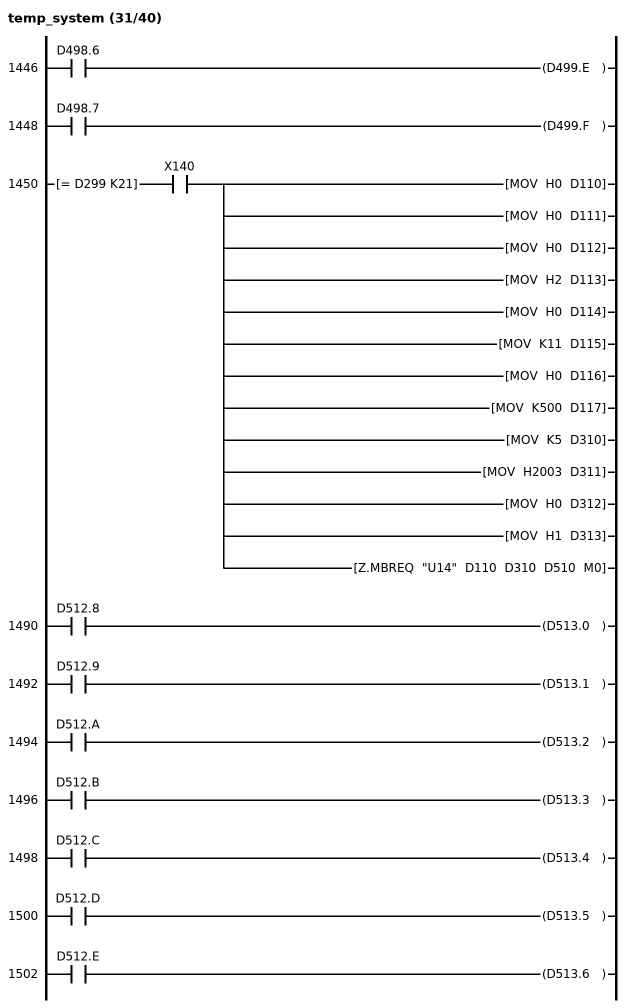
[picture p264: ladder of temp_system, rungs at steps 1446 to 1502]
1446  LD      D498.6
      OUT     D499.E
1448  LD      D498.7
      OUT     D499.F
1450  LD=     D299 K21
      AND     X140
      MOV     H0 D110
      MOV     H0 D111
      MOV     H0 D112
      MOV     H2 D113
      MOV     H0 D114
      MOV     K11 D115
      MOV     H0 D116
      MOV     K500 D117
      MOV     K5 D310
      MOV     H2003 D311
      MOV     H0 D312
      MOV     H1 D313
      Z.MBREQ "U14" D110 D310 D510 M0
1490  LD      D512.8
      OUT     D513.0
1492  LD      D512.9
      OUT     D513.1
1494  LD      D512.A
      OUT     D513.2
1496  LD      D512.B
      OUT     D513.3
1498  LD      D512.C
      OUT     D513.4
1500  LD      D512.D
      OUT     D513.5
1502  LD      D512.E
      OUT     D513.6
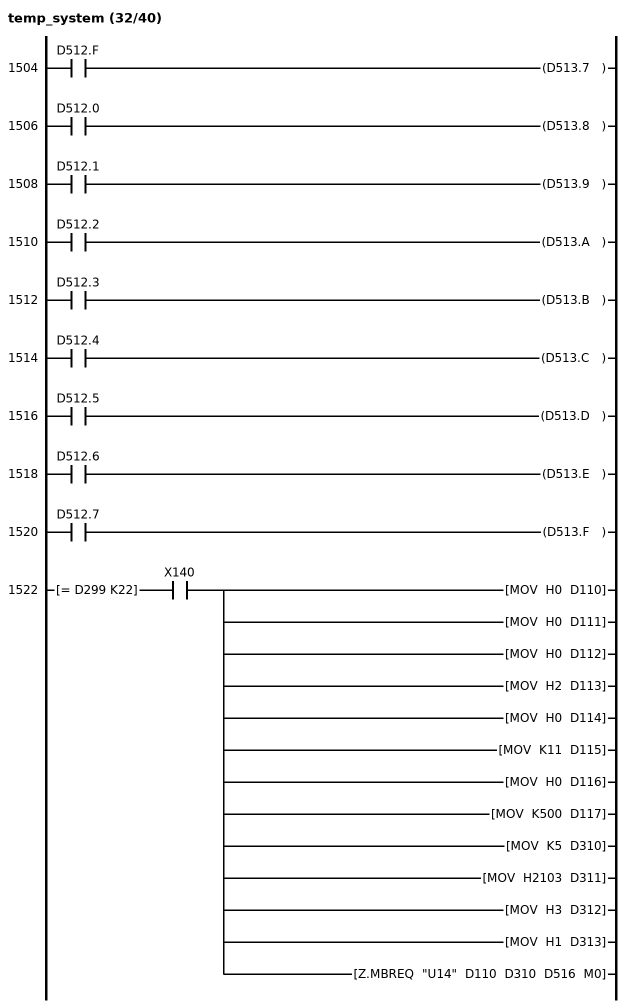
1504  LD      D512.F
      OUT     D513.7
1506  LD      D512.0
      OUT     D513.8
1508  LD      D512.1
      OUT     D513.9
1510  LD      D512.2
      OUT     D513.A
1512  LD      D512.3
      OUT     D513.B
1514  LD      D512.4
      OUT     D513.C
1516  LD      D512.5
      OUT     D513.D
1518  LD      D512.6
      OUT     D513.E
1520  LD      D512.7
      OUT     D513.F
1522  LD=     D299 K22
      AND     X140
      MOV     H0 D110
      MOV     H0 D111
      MOV     H0 D112
      MOV     H2 D113
      MOV     H0 D114
      MOV     K11 D115
      MOV     H0 D116
      MOV     K500 D117
      MOV     K5 D310
      MOV     H2103 D311
      MOV     H3 D312
      MOV     H1 D313
      Z.MBREQ "U14" D110 D310 D516 M0
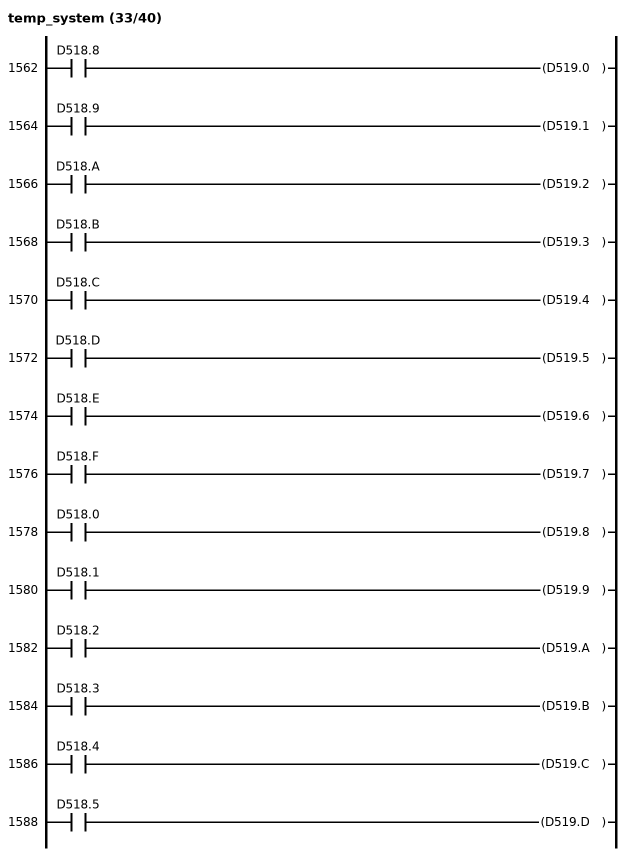
1562  LD      D518.8
      OUT     D519.0
1564  LD      D518.9
      OUT     D519.1
1566  LD      D518.A
      OUT     D519.2
1568  LD      D518.B
      OUT     D519.3
1570  LD      D518.C
      OUT     D519.4
1572  LD      D518.D
      OUT     D519.5
1574  LD      D518.E
      OUT     D519.6
1576  LD      D518.F
      OUT     D519.7
1578  LD      D518.0
      OUT     D519.8
1580  LD      D518.1
      OUT     D519.9
1582  LD      D518.2
      OUT     D519.A
1584  LD      D518.3
      OUT     D519.B
1586  LD      D518.4
      OUT     D519.C
1588  LD      D518.5
      OUT     D519.D
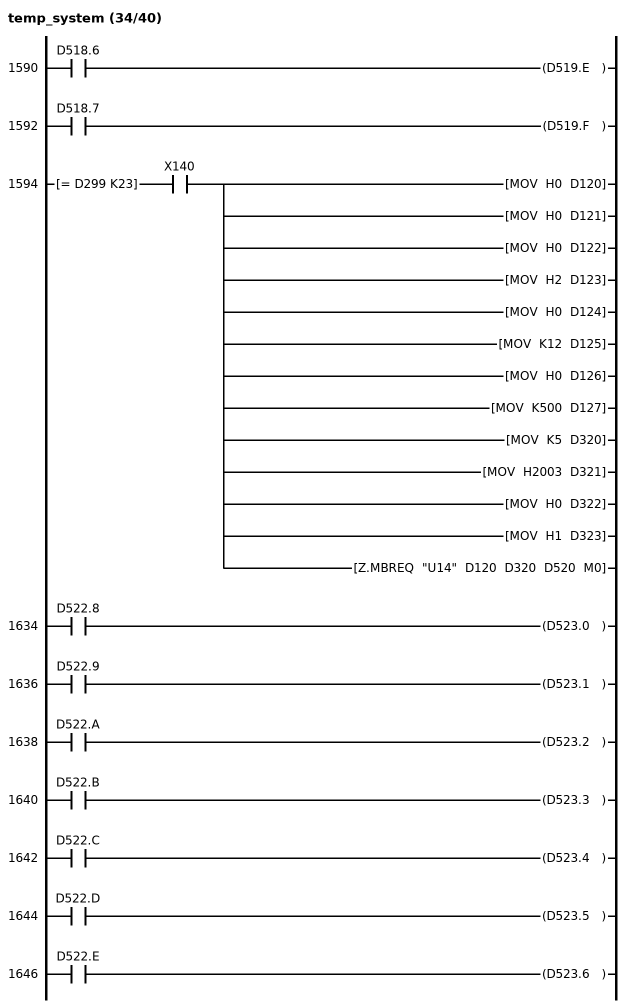
1590  LD      D518.6
      OUT     D519.E
1592  LD      D518.7
      OUT     D519.F
1594  LD=     D299 K23
      AND     X140
      MOV     H0 D120
      MOV     H0 D121
      MOV     H0 D122
      MOV     H2 D123
      MOV     H0 D124
      MOV     K12 D125
      MOV     H0 D126
      MOV     K500 D127
      MOV     K5 D320
      MOV     H2003 D321
      MOV     H0 D322
      MOV     H1 D323
      Z.MBREQ "U14" D120 D320 D520 M0
1634  LD      D522.8
      OUT     D523.0
1636  LD      D522.9
      OUT     D523.1
1638  LD      D522.A
      OUT     D523.2
1640  LD      D522.B
      OUT     D523.3
1642  LD      D522.C
      OUT     D523.4
1644  LD      D522.D
      OUT     D523.5
1646  LD      D522.E
      OUT     D523.6
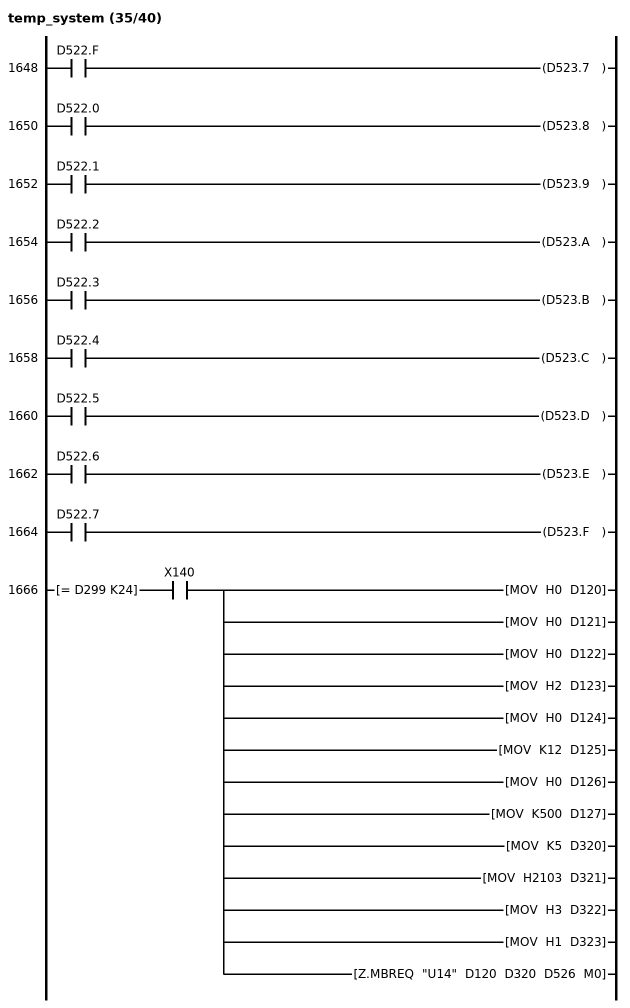
1648  LD      D522.F
      OUT     D523.7
1650  LD      D522.0
      OUT     D523.8
1652  LD      D522.1
      OUT     D523.9
1654  LD      D522.2
      OUT     D523.A
1656  LD      D522.3
      OUT     D523.B
1658  LD      D522.4
      OUT     D523.C
1660  LD      D522.5
      OUT     D523.D
1662  LD      D522.6
      OUT     D523.E
1664  LD      D522.7
      OUT     D523.F
1666  LD=     D299 K24
      AND     X140
      MOV     H0 D120
      MOV     H0 D121
      MOV     H0 D122
      MOV     H2 D123
      MOV     H0 D124
      MOV     K12 D125
      MOV     H0 D126
      MOV     K500 D127
      MOV     K5 D320
      MOV     H2103 D321
      MOV     H3 D322
      MOV     H1 D323
      Z.MBREQ "U14" D120 D320 D526 M0
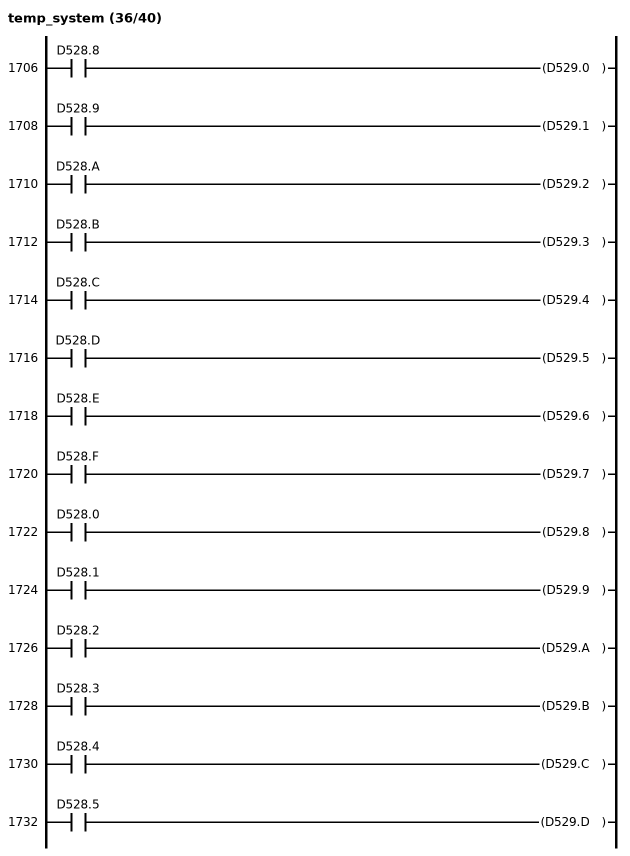
1706  LD      D528.8
      OUT     D529.0
1708  LD      D528.9
      OUT     D529.1
1710  LD      D528.A
      OUT     D529.2
1712  LD      D528.B
      OUT     D529.3
1714  LD      D528.C
      OUT     D529.4
1716  LD      D528.D
      OUT     D529.5
1718  LD      D528.E
      OUT     D529.6
1720  LD      D528.F
      OUT     D529.7
1722  LD      D528.0
      OUT     D529.8
1724  LD      D528.1
      OUT     D529.9
1726  LD      D528.2
      OUT     D529.A
1728  LD      D528.3
      OUT     D529.B
1730  LD      D528.4
      OUT     D529.C
1732  LD      D528.5
      OUT     D529.D
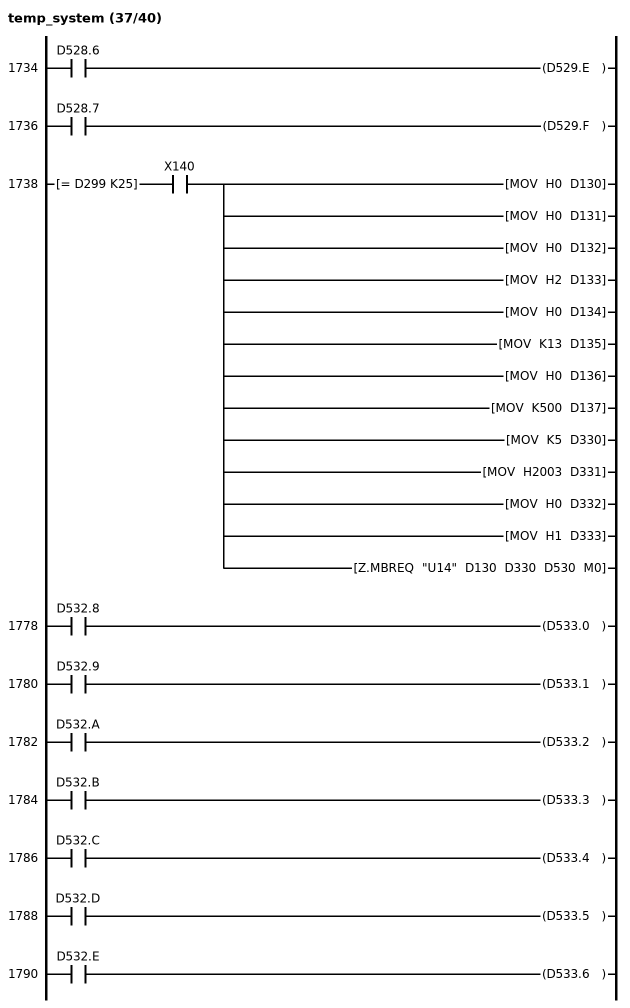
1734  LD      D528.6
      OUT     D529.E
1736  LD      D528.7
      OUT     D529.F
1738  LD=     D299 K25
      AND     X140
      MOV     H0 D130
      MOV     H0 D131
      MOV     H0 D132
      MOV     H2 D133
      MOV     H0 D134
      MOV     K13 D135
      MOV     H0 D136
      MOV     K500 D137
      MOV     K5 D330
      MOV     H2003 D331
      MOV     H0 D332
      MOV     H1 D333
      Z.MBREQ "U14" D130 D330 D530 M0
1778  LD      D532.8
      OUT     D533.0
1780  LD      D532.9
      OUT     D533.1
1782  LD      D532.A
      OUT     D533.2
1784  LD      D532.B
      OUT     D533.3
1786  LD      D532.C
      OUT     D533.4
1788  LD      D532.D
      OUT     D533.5
1790  LD      D532.E
      OUT     D533.6
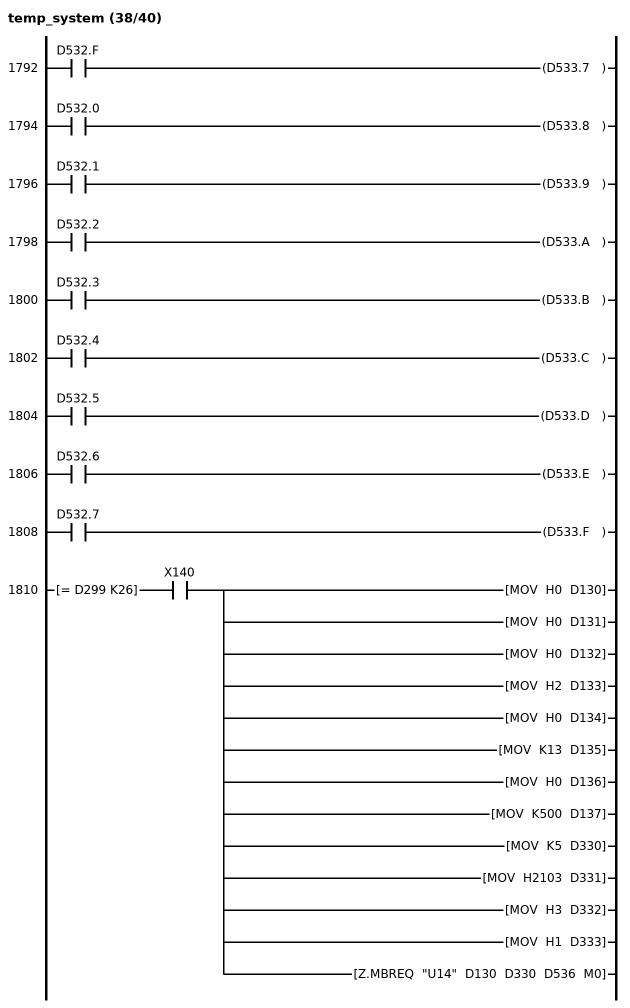
1792  LD      D532.F
      OUT     D533.7
1794  LD      D532.0
      OUT     D533.8
1796  LD      D532.1
      OUT     D533.9
1798  LD      D532.2
      OUT     D533.A
1800  LD      D532.3
      OUT     D533.B
1802  LD      D532.4
      OUT     D533.C
1804  LD      D532.5
      OUT     D533.D
1806  LD      D532.6
      OUT     D533.E
1808  LD      D532.7
      OUT     D533.F
1810  LD=     D299 K26
      AND     X140
      MOV     H0 D130
      MOV     H0 D131
      MOV     H0 D132
      MOV     H2 D133
      MOV     H0 D134
      MOV     K13 D135
      MOV     H0 D136
      MOV     K500 D137
      MOV     K5 D330
      MOV     H2103 D331
      MOV     H3 D332
      MOV     H1 D333
      Z.MBREQ "U14" D130 D330 D536 M0
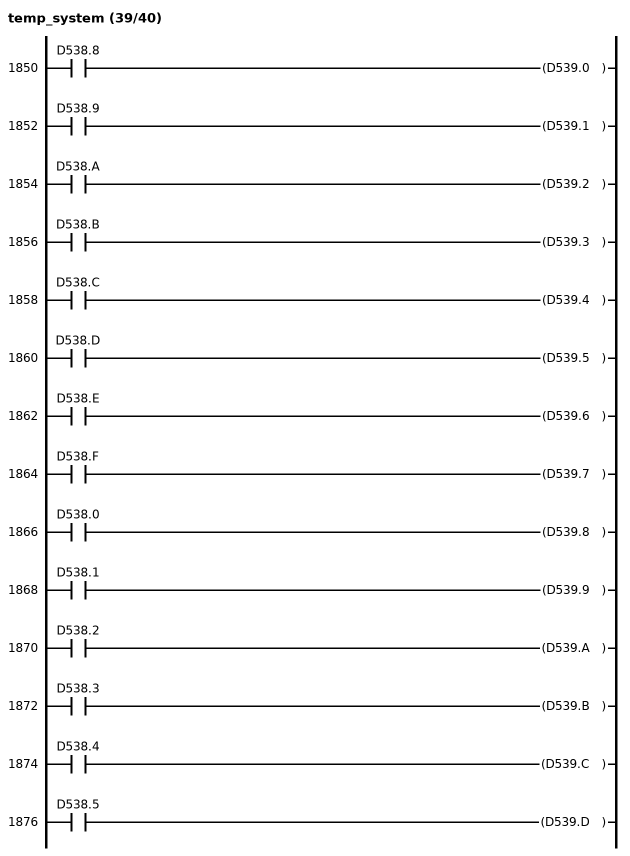
1850  LD      D538.8
      OUT     D539.0
1852  LD      D538.9
      OUT     D539.1
1854  LD      D538.A
      OUT     D539.2
1856  LD      D538.B
      OUT     D539.3
1858  LD      D538.C
      OUT     D539.4
1860  LD      D538.D
      OUT     D539.5
1862  LD      D538.E
      OUT     D539.6
1864  LD      D538.F
      OUT     D539.7
1866  LD      D538.0
      OUT     D539.8
1868  LD      D538.1
      OUT     D539.9
1870  LD      D538.2
      OUT     D539.A
1872  LD      D538.3
      OUT     D539.B
1874  LD      D538.4
      OUT     D539.C
1876  LD      D538.5
      OUT     D539.D
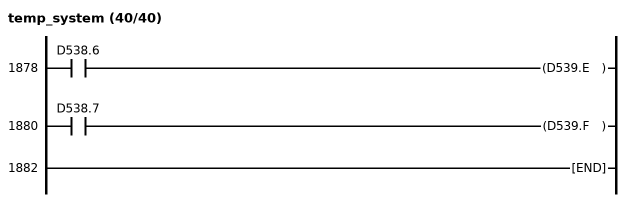
1878  LD      D538.6
      OUT     D539.E
1880  LD      D538.7
      OUT     D539.F
1882  END
END_PROGRAM

PROGRAM tempLOCK
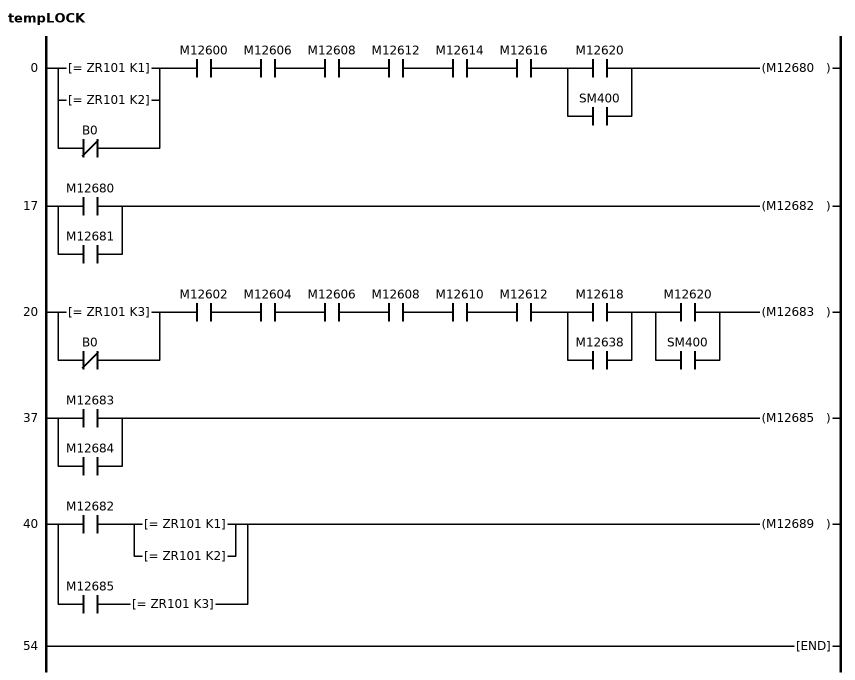
0     LD=     ZR101 K1
      OR=     ZR101 K2
      ORI     B0
      AND     M12600
      AND     M12606
      AND     M12608
      AND     M12612
      AND     M12614
      AND     M12616
      LD      M12620
      OR      SM400
      ANB
      OUT     M12680
17    LD      M12680
      OR      M12681
      OUT     M12682
20    LD=     ZR101 K3
      ORI     B0
      AND     M12602
      AND     M12604
      AND     M12606
      AND     M12608
      AND     M12610
      AND     M12612
      LD      M12618
      OR      M12638
      ANB
      LD      M12620
      OR      SM400
      ANB
      OUT     M12683
37    LD      M12683
      OR      M12684
      OUT     M12685
40    LD      M12682
      LD=     ZR101 K1
      OR=     ZR101 K2
      ANB
      LD      M12685
      AND=    ZR101 K3
      ORB
      OUT     M12689
54    END
END_PROGRAM

PROGRAM tower_lamp
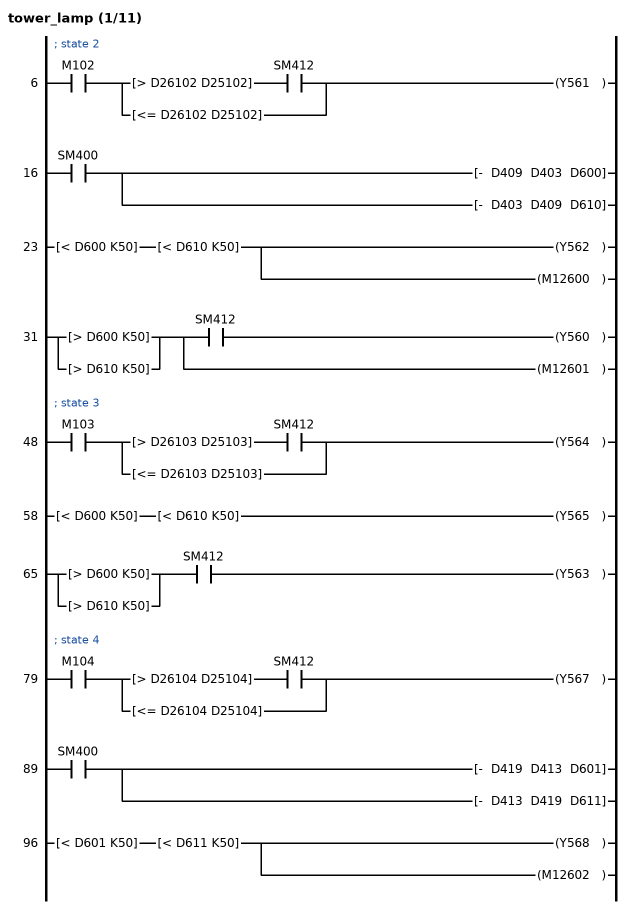
; state 2
6     LD      M102
      LD>     D26102 D25102
      AND     SM412
      OR<=    D26102 D25102
      ANB
      OUT     Y561
16    LD      SM400
      -       D409 D403 D600
      -       D403 D409 D610
23    LD<     D600 K50
      AND<    D610 K50
      OUT     Y562
      OUT     M12600
31    LD>     D600 K50
      OR>     D610 K50
      MPS
      AND     SM412
      OUT     Y560
      MPP
      OUT     M12601
; state 3
48    LD      M103
      LD>     D26103 D25103
      AND     SM412
      OR<=    D26103 D25103
      ANB
      OUT     Y564
58    LD<     D600 K50
      AND<    D610 K50
      OUT     Y565
65    LD>     D600 K50
      OR>     D610 K50
      AND     SM412
      OUT     Y563
; state 4
79    LD      M104
      LD>     D26104 D25104
      AND     SM412
      OR<=    D26104 D25104
      ANB
      OUT     Y567
89    LD      SM400
      -       D419 D413 D601
      -       D413 D419 D611
96    LD<     D601 K50
      AND<    D611 K50
      OUT     Y568
      OUT     M12602
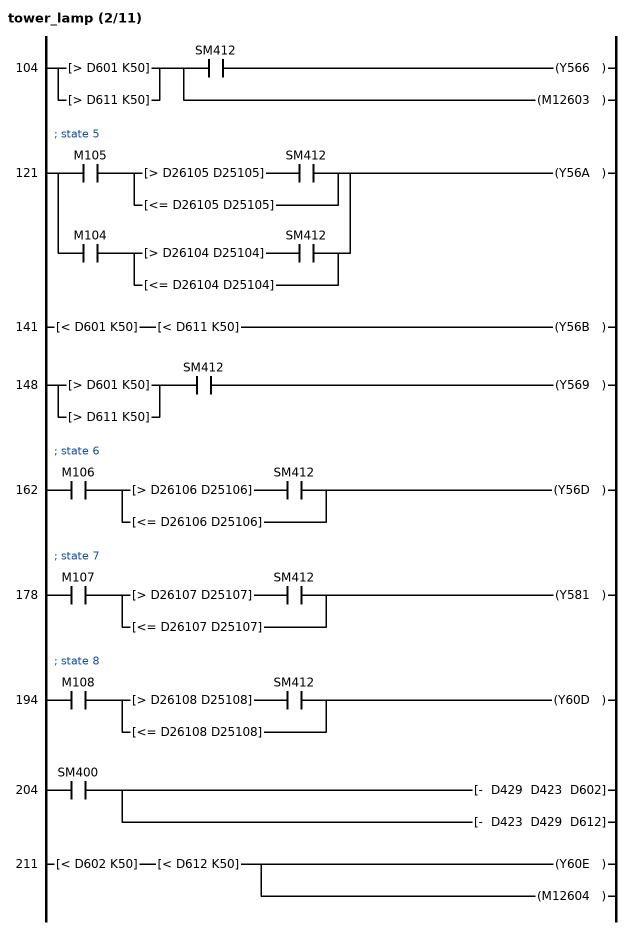
104   LD>     D601 K50
      OR>     D611 K50
      MPS
      AND     SM412
      OUT     Y566
      MPP
      OUT     M12603
; state 5
121   LD      M105
      LD>     D26105 D25105
      AND     SM412
      OR<=    D26105 D25105
      ANB
      LD      M104
      LD>     D26104 D25104
      AND     SM412
      OR<=    D26104 D25104
      ANB
      ORB
      OUT     Y56A
141   LD<     D601 K50
      AND<    D611 K50
      OUT     Y56B
148   LD>     D601 K50
      OR>     D611 K50
      AND     SM412
      OUT     Y569
; state 6
162   LD      M106
      LD>     D26106 D25106
      AND     SM412
      OR<=    D26106 D25106
      ANB
      OUT     Y56D
; state 7
178   LD      M107
      LD>     D26107 D25107
      AND     SM412
      OR<=    D26107 D25107
      ANB
      OUT     Y581
; state 8
194   LD      M108
      LD>     D26108 D25108
      AND     SM412
      OR<=    D26108 D25108
      ANB
      OUT     Y60D
204   LD      SM400
      -       D429 D423 D602
      -       D423 D429 D612
211   LD<     D602 K50
      AND<    D612 K50
      OUT     Y60E
      OUT     M12604
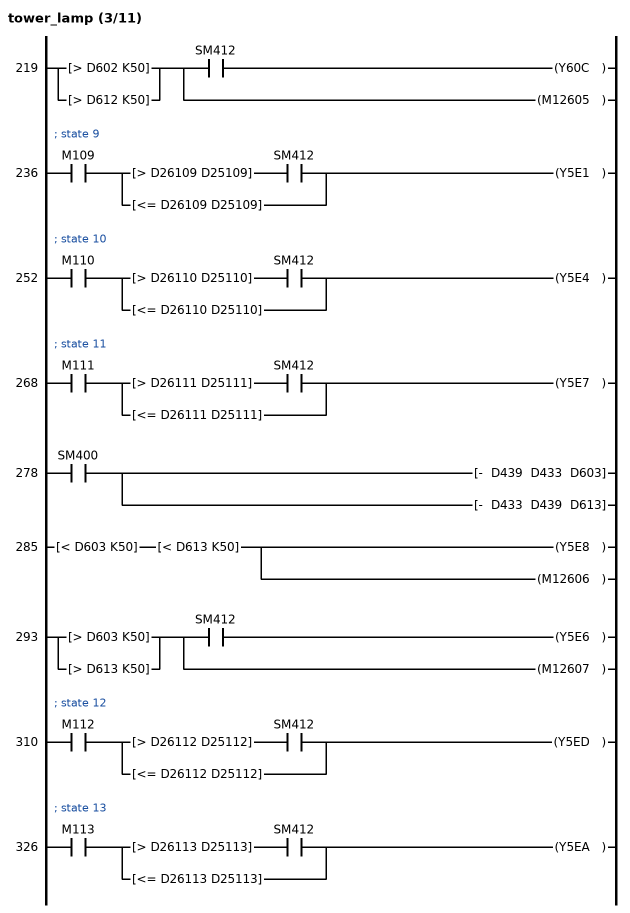
219   LD>     D602 K50
      OR>     D612 K50
      MPS
      AND     SM412
      OUT     Y60C
      MPP
      OUT     M12605
; state 9
236   LD      M109
      LD>     D26109 D25109
      AND     SM412
      OR<=    D26109 D25109
      ANB
      OUT     Y5E1
; state 10
252   LD      M110
      LD>     D26110 D25110
      AND     SM412
      OR<=    D26110 D25110
      ANB
      OUT     Y5E4
; state 11
268   LD      M111
      LD>     D26111 D25111
      AND     SM412
      OR<=    D26111 D25111
      ANB
      OUT     Y5E7
278   LD      SM400
      -       D439 D433 D603
      -       D433 D439 D613
285   LD<     D603 K50
      AND<    D613 K50
      OUT     Y5E8
      OUT     M12606
293   LD>     D603 K50
      OR>     D613 K50
      MPS
      AND     SM412
      OUT     Y5E6
      MPP
      OUT     M12607
; state 12
310   LD      M112
      LD>     D26112 D25112
      AND     SM412
      OR<=    D26112 D25112
      ANB
      OUT     Y5ED
; state 13
326   LD      M113
      LD>     D26113 D25113
      AND     SM412
      OR<=    D26113 D25113
      ANB
      OUT     Y5EA
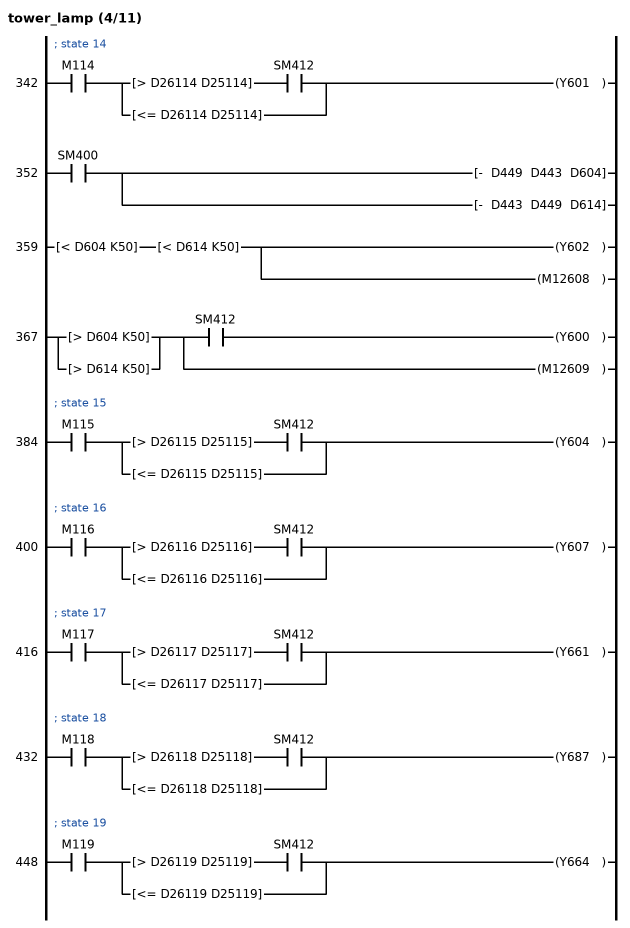
; state 14
342   LD      M114
      LD>     D26114 D25114
      AND     SM412
      OR<=    D26114 D25114
      ANB
      OUT     Y601
352   LD      SM400
      -       D449 D443 D604
      -       D443 D449 D614
359   LD<     D604 K50
      AND<    D614 K50
      OUT     Y602
      OUT     M12608
367   LD>     D604 K50
      OR>     D614 K50
      MPS
      AND     SM412
      OUT     Y600
      MPP
      OUT     M12609
; state 15
384   LD      M115
      LD>     D26115 D25115
      AND     SM412
      OR<=    D26115 D25115
      ANB
      OUT     Y604
; state 16
400   LD      M116
      LD>     D26116 D25116
      AND     SM412
      OR<=    D26116 D25116
      ANB
      OUT     Y607
; state 17
416   LD      M117
      LD>     D26117 D25117
      AND     SM412
      OR<=    D26117 D25117
      ANB
      OUT     Y661
; state 18
432   LD      M118
      LD>     D26118 D25118
      AND     SM412
      OR<=    D26118 D25118
      ANB
      OUT     Y687
; state 19
448   LD      M119
      LD>     D26119 D25119
      AND     SM412
      OR<=    D26119 D25119
      ANB
      OUT     Y664
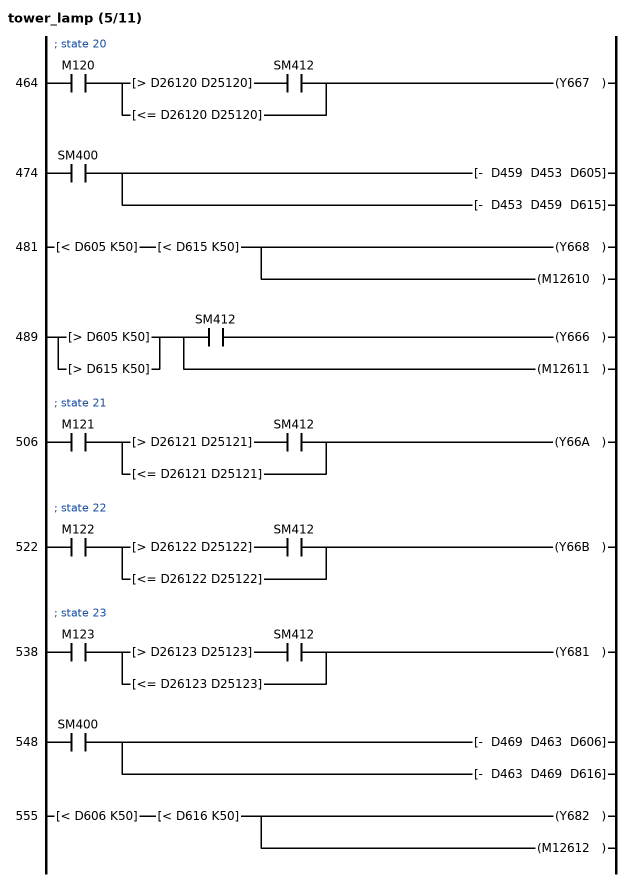
; state 20
464   LD      M120
      LD>     D26120 D25120
      AND     SM412
      OR<=    D26120 D25120
      ANB
      OUT     Y667
474   LD      SM400
      -       D459 D453 D605
      -       D453 D459 D615
481   LD<     D605 K50
      AND<    D615 K50
      OUT     Y668
      OUT     M12610
489   LD>     D605 K50
      OR>     D615 K50
      MPS
      AND     SM412
      OUT     Y666
      MPP
      OUT     M12611
; state 21
506   LD      M121
      LD>     D26121 D25121
      AND     SM412
      OR<=    D26121 D25121
      ANB
      OUT     Y66A
; state 22
522   LD      M122
      LD>     D26122 D25122
      AND     SM412
      OR<=    D26122 D25122
      ANB
      OUT     Y66B
; state 23
538   LD      M123
      LD>     D26123 D25123
      AND     SM412
      OR<=    D26123 D25123
      ANB
      OUT     Y681
548   LD      SM400
      -       D469 D463 D606
      -       D463 D469 D616
555   LD<     D606 K50
      AND<    D616 K50
      OUT     Y682
      OUT     M12612
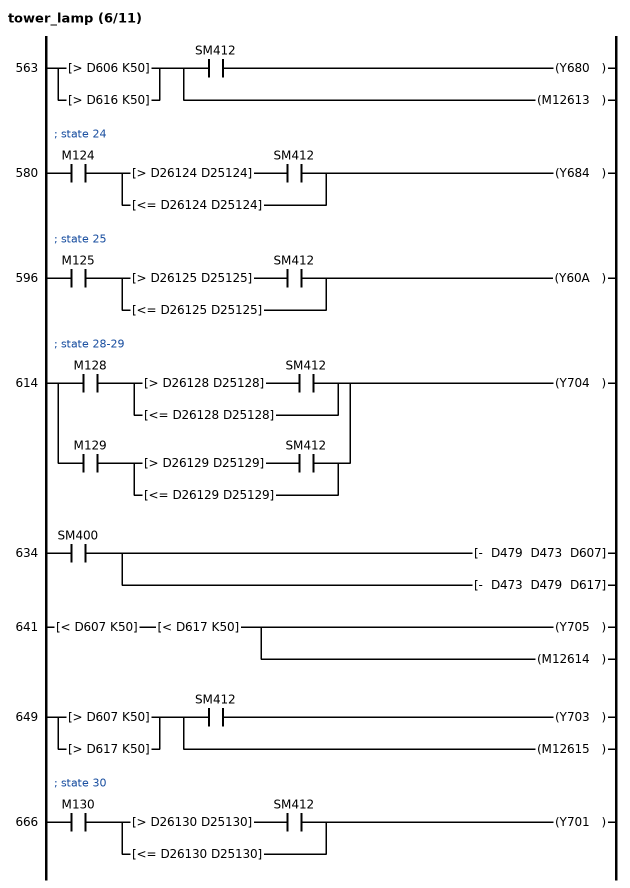
563   LD>     D606 K50
      OR>     D616 K50
      MPS
      AND     SM412
      OUT     Y680
      MPP
      OUT     M12613
; state 24
580   LD      M124
      LD>     D26124 D25124
      AND     SM412
      OR<=    D26124 D25124
      ANB
      OUT     Y684
; state 25
596   LD      M125
      LD>     D26125 D25125
      AND     SM412
      OR<=    D26125 D25125
      ANB
      OUT     Y60A
; state 28-29
614   LD      M128
      LD>     D26128 D25128
      AND     SM412
      OR<=    D26128 D25128
      ANB
      LD      M129
      LD>     D26129 D25129
      AND     SM412
      OR<=    D26129 D25129
      ANB
      ORB
      OUT     Y704
634   LD      SM400
      -       D479 D473 D607
      -       D473 D479 D617
641   LD<     D607 K50
      AND<    D617 K50
      OUT     Y705
      OUT     M12614
649   LD>     D607 K50
      OR>     D617 K50
      MPS
      AND     SM412
      OUT     Y703
      MPP
      OUT     M12615
; state 30
666   LD      M130
      LD>     D26130 D25130
      AND     SM412
      OR<=    D26130 D25130
      ANB
      OUT     Y701
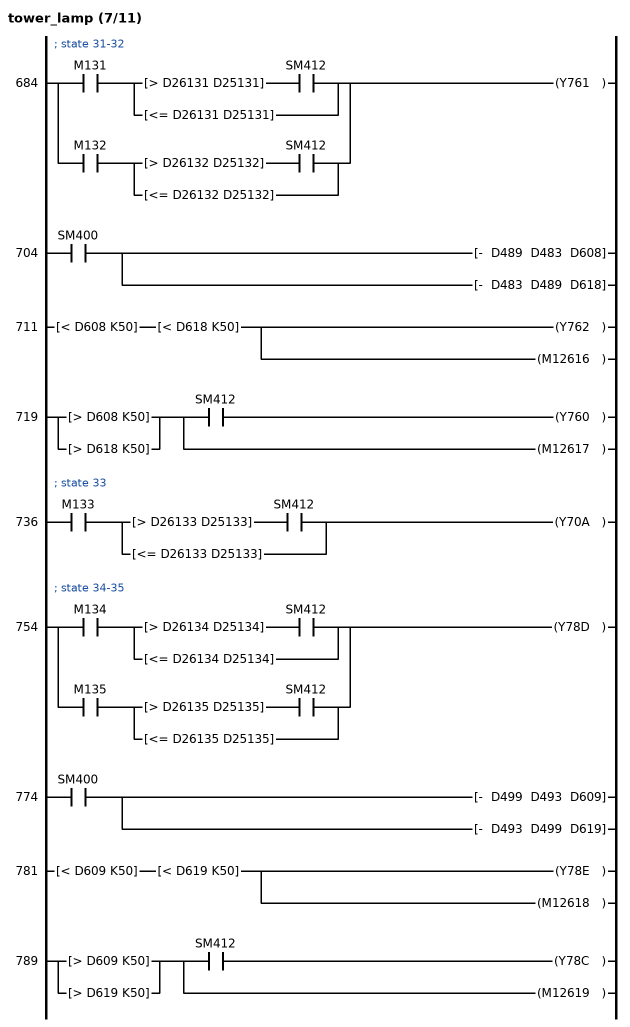
; state 31-32
684   LD      M131
      LD>     D26131 D25131
      AND     SM412
      OR<=    D26131 D25131
      ANB
      LD      M132
      LD>     D26132 D25132
      AND     SM412
      OR<=    D26132 D25132
      ANB
      ORB
      OUT     Y761
704   LD      SM400
      -       D489 D483 D608
      -       D483 D489 D618
711   LD<     D608 K50
      AND<    D618 K50
      OUT     Y762
      OUT     M12616
719   LD>     D608 K50
      OR>     D618 K50
      MPS
      AND     SM412
      OUT     Y760
      MPP
      OUT     M12617
; state 33
736   LD      M133
      LD>     D26133 D25133
      AND     SM412
      OR<=    D26133 D25133
      ANB
      OUT     Y70A
; state 34-35
754   LD      M134
      LD>     D26134 D25134
      AND     SM412
      OR<=    D26134 D25134
      ANB
      LD      M135
      LD>     D26135 D25135
      AND     SM412
      OR<=    D26135 D25135
      ANB
      ORB
      OUT     Y78D
774   LD      SM400
      -       D499 D493 D609
      -       D493 D499 D619
781   LD<     D609 K50
      AND<    D619 K50
      OUT     Y78E
      OUT     M12618
789   LD>     D609 K50
      OR>     D619 K50
      MPS
      AND     SM412
      OUT     Y78C
      MPP
      OUT     M12619
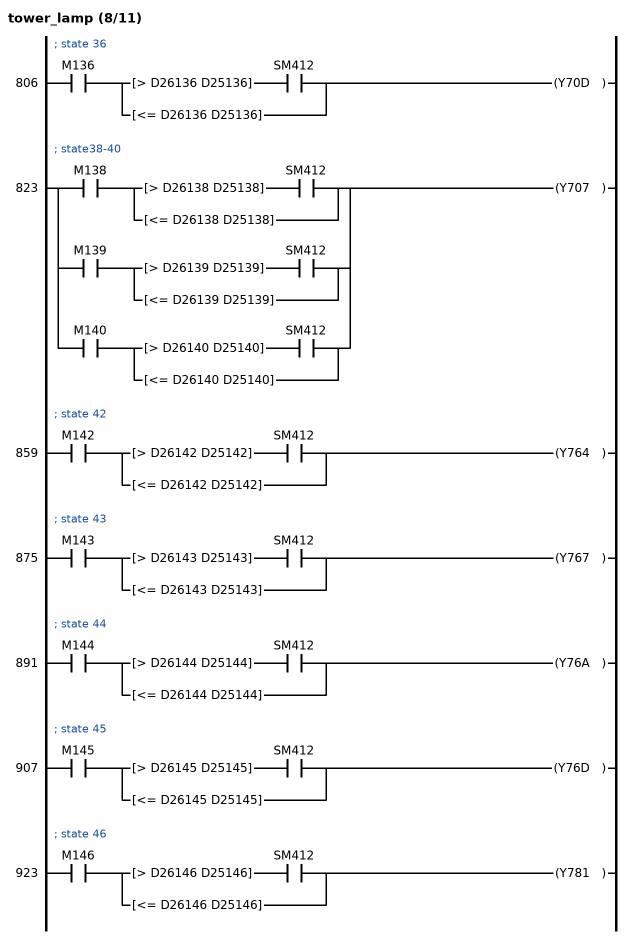
; state 36
806   LD      M136
      LD>     D26136 D25136
      AND     SM412
      OR<=    D26136 D25136
      ANB
      OUT     Y70D
; state38-40
823   LD      M138
      LD>     D26138 D25138
      AND     SM412
      OR<=    D26138 D25138
      ANB
      LD      M139
      LD>     D26139 D25139
      AND     SM412
      OR<=    D26139 D25139
      ANB
      ORB
      LD      M140
      LD>     D26140 D25140
      AND     SM412
      OR<=    D26140 D25140
      ANB
      ORB
      OUT     Y707
; state 42
859   LD      M142
      LD>     D26142 D25142
      AND     SM412
      OR<=    D26142 D25142
      ANB
      OUT     Y764
; state 43
875   LD      M143
      LD>     D26143 D25143
      AND     SM412
      OR<=    D26143 D25143
      ANB
      OUT     Y767
; state 44
891   LD      M144
      LD>     D26144 D25144
      AND     SM412
      OR<=    D26144 D25144
      ANB
      OUT     Y76A
; state 45
907   LD      M145
      LD>     D26145 D25145
      AND     SM412
      OR<=    D26145 D25145
      ANB
      OUT     Y76D
; state 46
923   LD      M146
      LD>     D26146 D25146
      AND     SM412
      OR<=    D26146 D25146
      ANB
      OUT     Y781
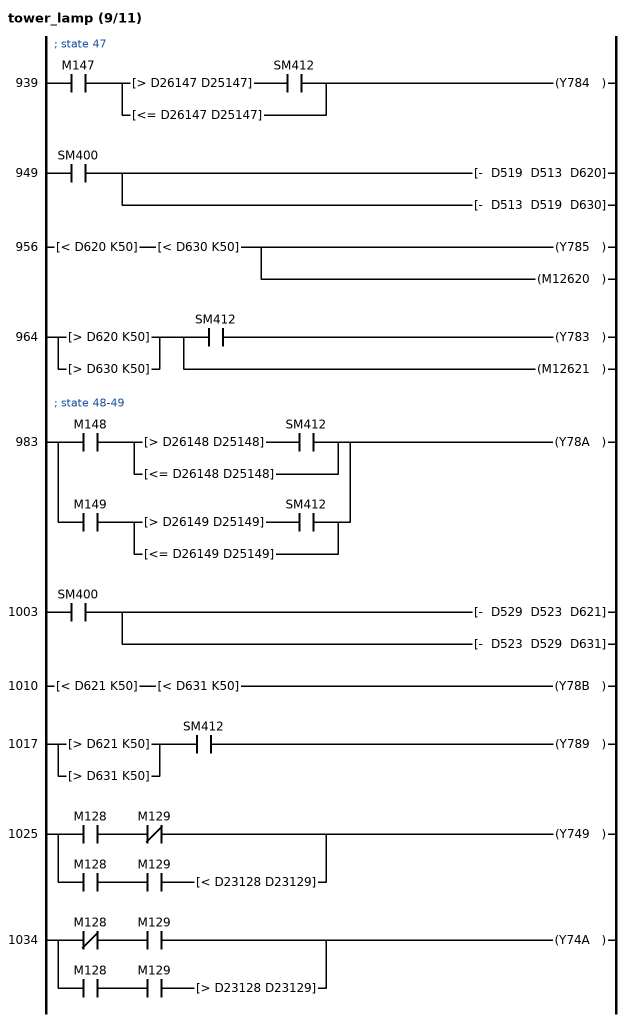
; state 47
939   LD      M147
      LD>     D26147 D25147
      AND     SM412
      OR<=    D26147 D25147
      ANB
      OUT     Y784
949   LD      SM400
      -       D519 D513 D620
      -       D513 D519 D630
956   LD<     D620 K50
      AND<    D630 K50
      OUT     Y785
      OUT     M12620
964   LD>     D620 K50
      OR>     D630 K50
      MPS
      AND     SM412
      OUT     Y783
      MPP
      OUT     M12621
; state 48-49
983   LD      M148
      LD>     D26148 D25148
      AND     SM412
      OR<=    D26148 D25148
      ANB
      LD      M149
      LD>     D26149 D25149
      AND     SM412
      OR<=    D26149 D25149
      ANB
      ORB
      OUT     Y78A
1003  LD      SM400
      -       D529 D523 D621
      -       D523 D529 D631
1010  LD<     D621 K50
      AND<    D631 K50
      OUT     Y78B
1017  LD>     D621 K50
      OR>     D631 K50
      AND     SM412
      OUT     Y789
1025  LD      M128
      ANI     M129
      LD      M128
      AND     M129
      AND<    D23128 D23129
      ORB
      OUT     Y749
1034  LDI     M128
      AND     M129
      LD      M128
      AND     M129
      AND>    D23128 D23129
      ORB
      OUT     Y74A
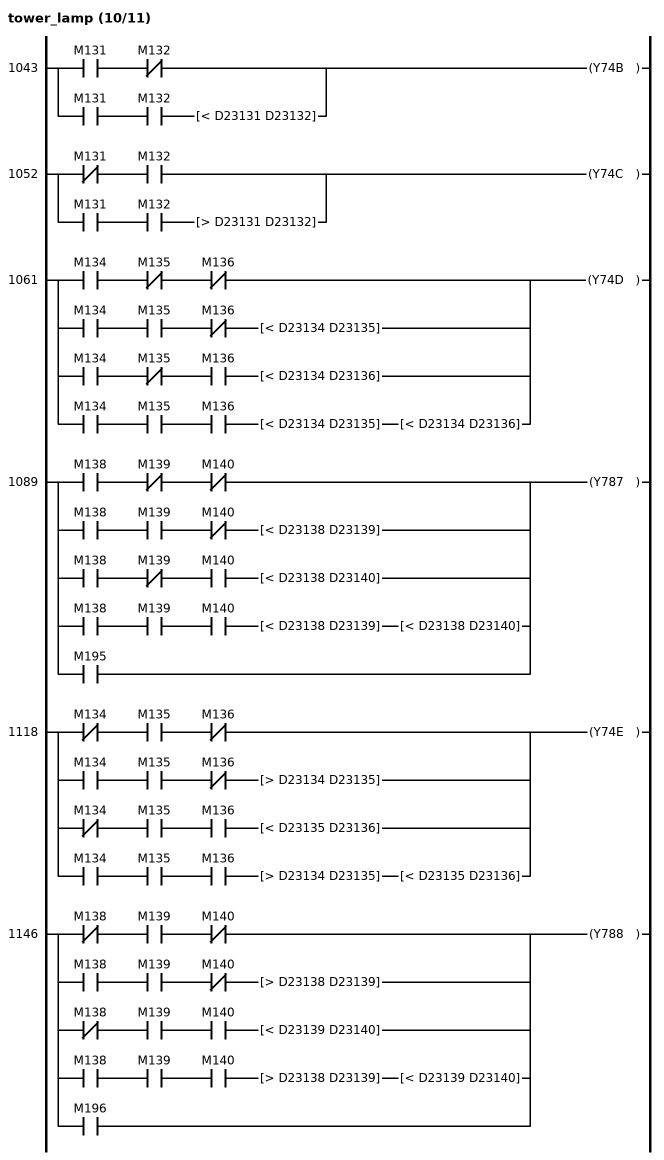
1043  LD      M131
      ANI     M132
      LD      M131
      AND     M132
      AND<    D23131 D23132
      ORB
      OUT     Y74B
1052  LDI     M131
      AND     M132
      LD      M131
      AND     M132
      AND>    D23131 D23132
      ORB
      OUT     Y74C
1061  LD      M134
      ANI     M135
      ANI     M136
      LD      M134
      AND     M135
      ANI     M136
      AND<    D23134 D23135
      ORB
      LD      M134
      ANI     M135
      AND     M136
      AND<    D23134 D23136
      ORB
      LD      M134
      AND     M135
      AND     M136
      AND<    D23134 D23135
      AND<    D23134 D23136
      ORB
      OUT     Y74D
1089  LD      M138
      ANI     M139
      ANI     M140
      LD      M138
      AND     M139
      ANI     M140
      AND<    D23138 D23139
      ORB
      LD      M138
      ANI     M139
      AND     M140
      AND<    D23138 D23140
      ORB
      LD      M138
      AND     M139
      AND     M140
      AND<    D23138 D23139
      AND<    D23138 D23140
      ORB
      OR      M195
      OUT     Y787
1118  LDI     M134
      AND     M135
      ANI     M136
      LD      M134
      AND     M135
      ANI     M136
      AND>    D23134 D23135
      ORB
      LDI     M134
      AND     M135
      AND     M136
      AND<    D23135 D23136
      ORB
      LD      M134
      AND     M135
      AND     M136
      AND>    D23134 D23135
      AND<    D23135 D23136
      ORB
      OUT     Y74E
1146  LDI     M138
      AND     M139
      ANI     M140
      LD      M138
      AND     M139
      ANI     M140
      AND>    D23138 D23139
      ORB
      LDI     M138
      AND     M139
      AND     M140
      AND<    D23139 D23140
      ORB
      LD      M138
      AND     M139
      AND     M140
      AND>    D23138 D23139
      AND<    D23139 D23140
      ORB
      OR      M196
      OUT     Y788
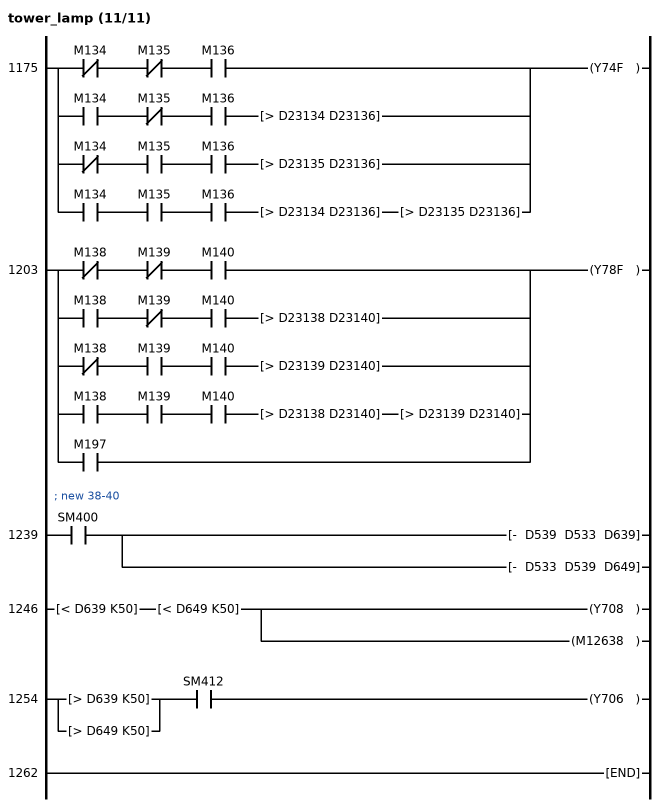
1175  LDI     M134
      ANI     M135
      AND     M136
      LD      M134
      ANI     M135
      AND     M136
      AND>    D23134 D23136
      ORB
      LDI     M134
      AND     M135
      AND     M136
      AND>    D23135 D23136
      ORB
      LD      M134
      AND     M135
      AND     M136
      AND>    D23134 D23136
      AND>    D23135 D23136
      ORB
      OUT     Y74F
1203  LDI     M138
      ANI     M139
      AND     M140
      LD      M138
      ANI     M139
      AND     M140
      AND>    D23138 D23140
      ORB
      LDI     M138
      AND     M139
      AND     M140
      AND>    D23139 D23140
      ORB
      LD      M138
      AND     M139
      AND     M140
      AND>    D23138 D23140
      AND>    D23139 D23140
      ORB
      OR      M197
      OUT     Y78F
; new 38-40
1239  LD      SM400
      -       D539 D533 D639
      -       D533 D539 D649
1246  LD<     D639 K50
      AND<    D649 K50
      OUT     Y708
      OUT     M12638
1254  LD>     D639 K50
      OR>     D649 K50
      AND     SM412
      OUT     Y706
1262  END
END_PROGRAM

PROGRAM tranverser
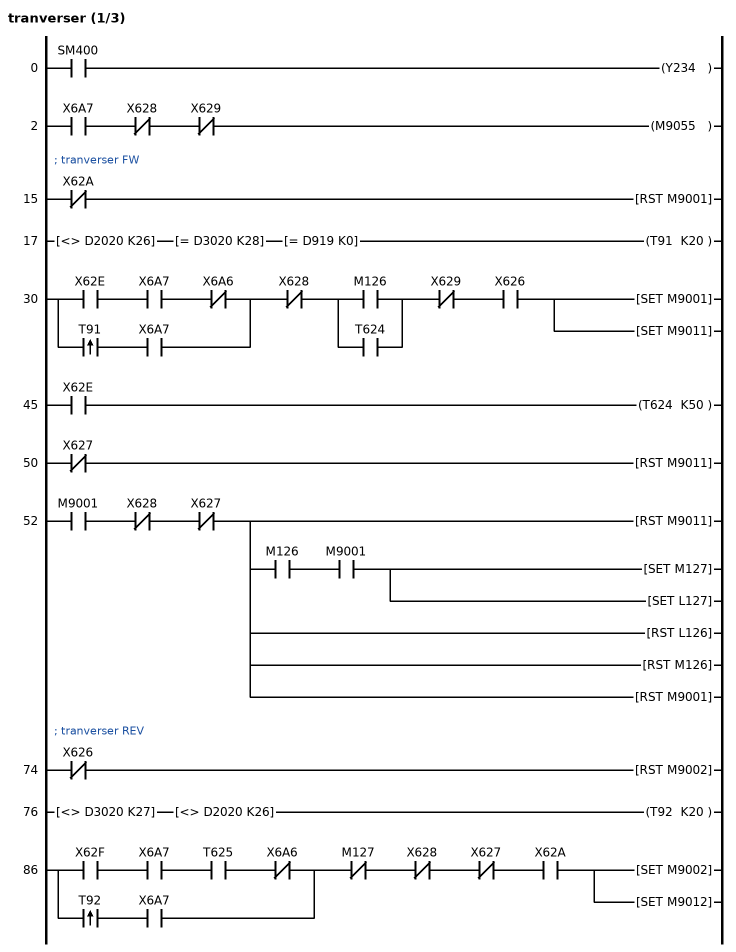
0     LD      SM400
      OUT     Y234
2     LD      X6A7
      ANI     X628
      ANI     X629
      OUT     M9055
; tranverser FW
15    LDI     X62A
      RST     M9001
17    LD<>    D2020 K26
      AND=    D3020 K28
      AND=    D919 K0
      OUT     T91 K20
30    LD      X62E
      AND     X6A7
      ANI     X6A6
      LDP     T91
      AND     X6A7
      ORB
      ANI     X628
      LD      M126
      OR      T624
      ANB
      ANI     X629
      AND     X626
      SET     M9001
      SET     M9011
45    LD      X62E
      OUT     T624 K50
50    LDI     X627
      RST     M9011
52    LD      M9001
      ANI     X628
      ANI     X627
      RST     M9011
      MPS
      AND     M126
      AND     M9001
      SET     M127
      SET     L127
      MPP
      RST     L126
      RST     M126
      RST     M9001
; tranverser REV
74    LDI     X626
      RST     M9002
76    LD<>    D3020 K27
      AND<>   D2020 K26
      OUT     T92 K20
86    LD      X62F
      AND     X6A7
      AND     T625
      ANI     X6A6
      LDP     T92
      AND     X6A7
      ORB
      ANI     M127
      ANI     X628
      ANI     X627
      AND     X62A
      SET     M9002
      SET     M9012
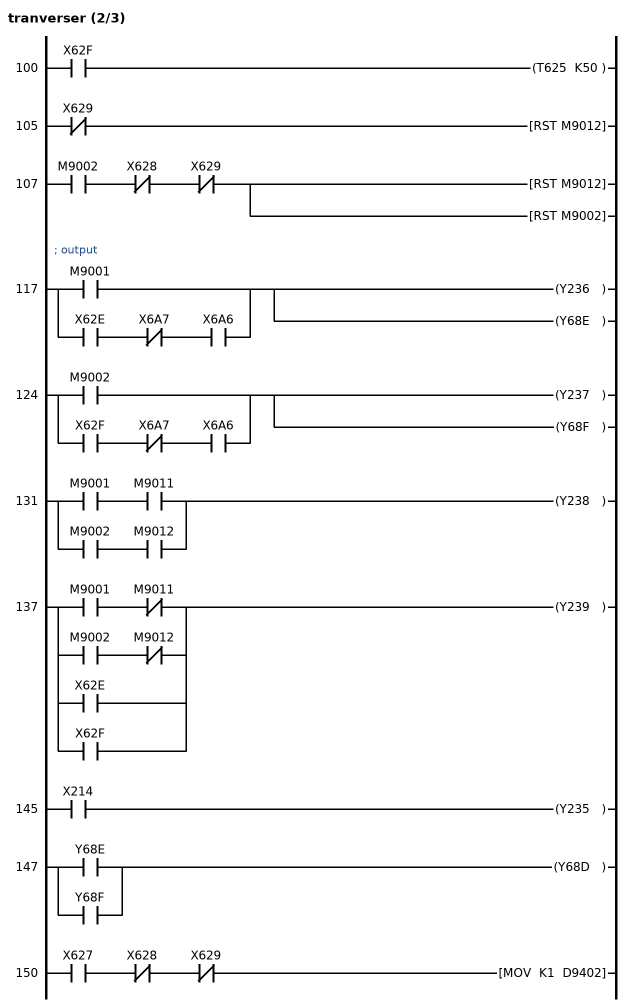
100   LD      X62F
      OUT     T625 K50
105   LDI     X629
      RST     M9012
107   LD      M9002
      ANI     X628
      ANI     X629
      RST     M9012
      RST     M9002
; output
117   LD      M9001
      LD      X62E
      ANI     X6A7
      AND     X6A6
      ORB
      OUT     Y236
      OUT     Y68E
124   LD      M9002
      LD      X62F
      ANI     X6A7
      AND     X6A6
      ORB
      OUT     Y237
      OUT     Y68F
131   LD      M9001
      AND     M9011
      LD      M9002
      AND     M9012
      ORB
      OUT     Y238
137   LD      M9001
      ANI     M9011
      LD      M9002
      ANI     M9012
      ORB
      OR      X62E
      OR      X62F
      OUT     Y239
145   LD      X214
      OUT     Y235
147   LD      Y68E
      OR      Y68F
      OUT     Y68D
150   LD      X627
      ANI     X628
      ANI     X629
      MOV     K1 D9402
